FUNCTION_BLOCK FB_SetChamberPressure
VAR_IN_OUT
	chamber	: ST_Volume;
END_VAR
VAR_INPUT
	rNewPressure	: REAL;
	Override	: BOOL :=FALSE;
END_VAR
VAR_OUTPUT
END_VAR
VAR
END_VAR

//If override boolean is on then set camber pressure to new pressure
IF Override THEN
	chamber.rPressure := rNewPressure;
END_IF

END_FUNCTION_BLOCK

(* stored: Version 1.1.0.1, ProductVersion 3.1.4020.12
   POU FB_SetChamberPressure: Id {9a121830-c1f4-44cb-9d10-7af373b6751a}, SpecialFunc None *)
